// TIA Portal V15 export
// export: Created 2019-02-11T17:35:21.1491863Z, ExportSetting WithDefaults, WithReadOnly, DisplayName Totally Integrated Automation Portal, DisplayVersion V15 Update 2, DisplayName TIA Portal Openness, DisplayVersion V15 Update 2, DisplayName STEP 7 Professional, DisplayVersion V15 Update 2, DisplayName STEP 7 Safety, DisplayVersion V15, DisplayName WinCC Professional, DisplayVersion V15 Update 2, DisplayName SIMATIC Visualization Architect, DisplayVersion V15 Update 1
DATA_BLOCK "FGDB_ROBNAME@Quiss"   // DB35
{ S7_Optimized_Access := 'FALSE' }
AUTHOR : integra
FAMILY : SUB
VERSION : 1.0
// stored: AutoNumber true, CodeModifiedDate 2019-02-11T17:31:31.2321174Z, CompileDate 2019-02-11T17:35:11.3309796Z, CreationDate 2019-02-11T17:31:31.1508364Z, DBAccessibleFromOPCUA true, InstanceOfName iSF_TECH_ROBOT_SEAM_INSPECTION, InstanceOfNumber 20, InstanceOfType FB, InterfaceModifiedDate 2018-01-31T08:44:02.5069254Z, IsConsistent true, IsKnowHowProtected false, ModifiedDate 2019-02-11T17:31:31.2321174Z, ParameterModified 2017-11-28T13:33:30.143072Z, StructureModified 2018-01-31T08:44:02.5069254Z, UDAEnableTagReadback false
"iSF_TECH_ROBOT_SEAM_INSPECTION"
   // VAR_INPUT
   //    fct : Int;
   //    resetResult : Bool;
   //    safetyStop : Bool;
   //    readyTarget : Bool;
   // END_VAR
   // VAR_OUTPUT
   //    resultOK : Bool;
   //    resultNOK : Bool;
   //    startTarget : Bool;
   //    fault : Bool;
   // END_VAR
   // VAR_IN_OUT
   //    IfcFGExternal : "iUDT_IFC_SYS_EXTERNAL_ALARM";
   //    IfcTECH : "iUDT_IFC_ROBOT_TECH";
   //    In_PI_TECH : "iUDT_PI_ROBOT_ADRxx48_TECH";
   //    OUT_PO_TECH : "iUDT_PO_ROBOT_ADRxx48_TECH";
   // END_VAR
   // VAR
   //    F : Struct
   //       wrongID : Bool;
   //       productError : Bool;
   //       resultNOK : Bool;
   //       targetNOK : Bool;
   //    END_STRUCT;
   //    Masks : Struct
   //       disableFault1_8 : Byte;
   //       prodRelevantFault1_8 : Byte;
   //    END_STRUCT;
   //    LastState : Struct
   //       fault1_8 : Byte;
   //       warning_1_8 : Byte;
   //    END_STRUCT;
   //    Tmr : Struct
   //       s1 { S7_SetPoint := 'True'} : Int;
   //       a1 : Int;
   //    END_STRUCT;
   //    TmrB : Struct
   //       "1_EnableDelayTime" : Bool;
   //       "1_RunDelayTime" : Bool;
   //       "1_DoneDelayTime" : Bool;
   //    END_STRUCT;
   //    D : Struct
   //       resultOK : Bool;
   //       resultNOK : Bool;
   //       fm_startTargetMesurment : Bool;
   //       fm_stopTargetMesurment : Bool;
   //       HM_StartTarget { ExternalAccessible := 'False'; ExternalVisible := 'False'; ExternalWritable := 'False'} : Bool;
   //       resetResult : Bool;
   //    END_STRUCT;
   //    VCB : Struct
   //       startTarget : Bool;
   //       stopTarget : Bool;
   //    END_STRUCT;
   //    Target : Struct
   //       SO_active : Bool;
   //       MO_active : Bool;
   //       TU_active : Bool;
   //       WE_active : Bool;
   //       TH_active : Bool;
   //       FR_active : Bool;
   //       SA_active : Bool;
   //       SO_HOUR : USInt;
   //       SO_MIN : USInt;
   //       MO_HOUR : USInt;
   //       MO_MIN : USInt;
   //       TU_HOUR : USInt;
   //       TU_MIN : USInt;
   //       WE_HOUR : USInt;
   //       WE_MIN : USInt;
   //       TH_HOUR : USInt;
   //       TH_MIN : USInt;
   //       FR_HOUR : USInt;
   //       FR_MIN : USInt;
   //       SA_HOUR : USInt;
   //       SA_MIN : USInt;
   //    END_STRUCT;
   //    TECH_IN : Struct
   //       ID : Byte;
   //       technoBit1 : Bool;
   //       technoBit2 : Bool;
   //       technoBit3 : Bool;
   //       technoBit4 : Bool;
   //       technoBit5 : Bool;
   //       technoBit6 : Bool;
   //       technoBit7 : Bool;
   //       technoBit8 : Bool;
   //       technoBit9 : Bool;
   //       technoBit10 : Bool;
   //       technoBit11 : Bool;
   //       technoBit12 : Bool;
   //       technoBit13 : Bool;
   //       technoBit14 : Bool;
   //       technoBit15 : Bool;
   //       technoBit16 : Bool;
   //       technoBit17 : Bool;
   //       technoBit18 : Bool;
   //       technoBit19 : Bool;
   //       technoBit20 : Bool;
   //       technoBit21 : Bool;
   //       technoBit22 : Bool;
   //       technoBit23 : Bool;
   //       technoBit24 : Bool;
   //       productOnOff : Bool;
   //       inspectionOnOff : Bool;
   //       systemReady : Bool;
   //       automaticReady : Bool;
   //       productSelectable : Bool;
   //       inspectionChangeable : Bool;
   //       resultAvaible : Bool;
   //       productResultOK : Bool;
   //       productResultWARNING : Bool;
   //       productResultNOK : Bool;
   //       productResultERROR : Bool;
   //       evaluationCompleted : Bool;
   //       technoBit37 : Bool;
   //       technoBit38 : Bool;
   //       technoBit39 : Bool;
   //       available : Bool;
   //    END_STRUCT;
   //    TECH_OUT : Struct
   //       ID : Byte;
   //       technoBit1 : Bool;
   //       technoBit2 : Bool;
   //       technoBit3 : Bool;
   //       technoBit4 : Bool;
   //       technoBit5 : Bool;
   //       technoBit6 : Bool;
   //       technoBit7 : Bool;
   //       technoBit8 : Bool;
   //       technoBit9 : Bool;
   //       technoBit10 : Bool;
   //       technoBit11 : Bool;
   //       technoBit12 : Bool;
   //       technoBit13 : Bool;
   //       technoBit14 : Bool;
   //       technoBit15 : Bool;
   //       technoBit16 : Bool;
   //       technoBit17 : Bool;
   //       technoBit18 : Bool;
   //       technoBit19 : Bool;
   //       technoBit20 : Bool;
   //       technoBit21 : Bool;
   //       technoBit22 : Bool;
   //       technoBit23 : Bool;
   //       technoBit24 : Bool;
   //       resetMeasurementResults : Bool;
   //       technoBit26 : Bool;
   //       technoBit27 : Bool;
   //       technoBit28 : Bool;
   //       technoBit29 : Bool;
   //       technoBit30 : Bool;
   //       technoBit31 : Bool;
   //       technoBit32 : Bool;
   //       technoBit33 : Bool;
   //       technoBit34 : Bool;
   //       technoBit35 : Bool;
   //       technoBit36 : Bool;
   //       technoBit37 : Bool;
   //       technoBit38 : Bool;
   //       technoBit39 : Bool;
   //       technoBit40 : Bool;
   //    END_STRUCT;
   // END_VAR
BEGIN
END_DATA_BLOCK
